// TIA Portal V20 export
// export: Created 2025-12-01T14:57:18.5462743Z, ExportSetting None, DisplayName Totally Integrated Automation Portal, DisplayVersion V20 Update 3, DisplayName TIA Portal Openness, DisplayVersion V20 Update 3, DisplayName TIA Portal Version Control Interface, DisplayVersion V20 Update 3, DisplayName STEP 7 Professional, DisplayVersion V20 Update 3, DisplayName STEP 7 Safety, DisplayVersion V20 Update 2, DisplayName WinCC Basic/Comfort/Advanced, DisplayVersion V20 Update 3, DisplayName WinCC Professional, DisplayVersion V20 Update 3, DisplayName WinCC Unified, DisplayVersion V20 Update 3
DATA_BLOCK "DB816_UTs_TextoPantalla"   // DB816
{ S7_Optimized_Access := 'FALSE' }
AUTHOR : TRACKING
NAME : 20130301
VERSION : 3.0
// stored: AutoNumber false
   VAR
      UT { S7_SetPoint := 'True'} : Array[0.."CTE_MaxUTs"] of "UDT_UTs_TextoPantalla";   // Array de UT's - Ruta de la UT
   END_VAR
BEGIN
END_DATA_BLOCK
